(* Logix 5000 project; controller DUNEW2PLC1 vendor 1 type 14 code 221 rev 33.11; software revision 33.00 *)

TASK DUNEWINDER2 (continuous, watchdog 500 ms) : main, state_9_unservo, state_11_eot_trip, state_10_error, state_6_latch, state_3_move_xy, state_5_move_z, state_1_ready, tension_pid, queued_motion, state_12_move_xz, state_13_move_yz, state_14_hmi_stop
TASK SafetyTask (periodic, rate 20 ms, priority 10, watchdog 20 ms) : Safety

MODULES
   Local : vendor 1 type 14 code 221 (5069 0, rev 33.11)
      DUNEW2AMP : 2198-P031 (Ethernet 192.168.140.15, rev 11.3, A_MotionDiagnostics RPI 1 ms, B_MotionSync RPI 2 ms)
      DUNEW2SERVO1 : vendor 1 type 45 code 31 (Ethernet 192.168.140.16, rev 11.3, C_Safety_Output RPI 20 ms, A_MotionDiagnostics RPI 1 ms, D_Safety_Input RPI 10 ms, B_MotionSync RPI 2 ms)
      DUNEW2SERVO2 : vendor 1 type 45 code 31 (Ethernet 192.168.140.17, rev 11.2, A_MotionDiagnostics RPI 1 ms, C_Safety_Output RPI 20 ms, B_MotionSync RPI 2 ms, D_Safety_Input RPI 10 ms)
      DUNEW2NETSW : vendor 1 type 12 code 241 (Ethernet 192.168.140.10, rev 10.1, Output RPI 1000 ms)
      DUNE2CAM1 : vendor 678 type 100 code 274 (Ethernet 192.168.140.19, rev 11.1, Output RPI 60 ms)
       : 5069-IB16 (5069 1, rev 2.14, StandardDataDriven RPI 5 ms)
           Local:1:I.Pt15.Data   // The wire break switch was causing electrical problems, so we use the load-cell as a proxy for wire break
           Local:1:I.Pt09.Data   // Latch middle
           Local:1:I.Pt08.Data   // Latch top
       : 5069-IB16 (5069 6, rev 2.14, StandardDataDriven RPI 5 ms)
       : 5069-IB16 (5069 2, rev 2.14, StandardDataDriven RPI 5 ms)
           Local:2:I.Pt07.Data   // O/T SWITCH OVERTRAVEL SWITCH
           Local:2:I.Pt13.Data   // Cabinet lighted push button
           Local:2:I.Pt06.Data   // TENSION ON/OFF
       : vendor 1 type 115 code 313 (5069 5, rev 2.1, StandardDataDriven RPI 13.1 ms)
           Local:5:O.Ch00.Data   // Tension_Servo_CMD
       : 5069-OB16 (5069 3, rev 2.14, StandardDataDriven RPI 5 ms)
           Local:3:O.Pt01.Data   // Latching signal output
           Local:3:O.Pt11.Data   // Reset PB - Light
           Local:3:O.Pt15.Data   // Beacon - Sounder
           Local:3:O.Pt13.Data   // Beacon - Amber
           Local:3:O.Pt14.Data   // Beacon - Red
           Local:3:O.Pt12.Data   // Beacon - Green
       : 5069-OB16 (5069 7, rev 2.14, StandardDataDriven RPI 5 ms)
       : 5069-IF8 (5069 4, rev 2.11, StandardDataDriven RPI 12.5 ms)
           Local:4:I   // Wire tension (N)
      DUNEW2PLC2 : 1734-AENT (Ethernet 192.168.140.14, rev 6.12)
          : vendor 1 type 35 code 16 (PointIO 2, rev 2.1, Output RPI 20 ms, Input RPI 10 ms)
          : vendor 1 type 35 code 15 (PointIO 1, rev 2.1, Output RPI 20 ms, Input RPI 10 ms)
              DUNEW2PLC2:1:I.Pt03Data   // EStop Pullcord 1
              DUNEW2PLC2:1:I.Pt01Data   // LC OSS2
              DUNEW2PLC2:1:I.Pt00Data   // LC OSS1
              DUNEW2PLC2:1:I.Pt04Data   // EStop Pullcord 2
              DUNEW2PLC2:1:I.Pt02Data   // EStop Rack
              DUNEW2PLC2:1:I.Pt05Data   // Run Key
END_MODULES

TYPE MotionSeg :   // motion segments for move queue, lines or arcs
STRUCT
   Valid : BOOL;   // segment valid flag
   SegType : SINT;   // 1=line, 2=arc
   XY : REAL[2];   // end xy
   Speed : REAL;   // >0
   Accel : REAL;   // >0
   Decel : REAL;   // >0
   JerkAccel : REAL;
   JerkDecel : REAL;
   TermType : SINT;   // 0 to 6
   Seq : DINT;   // Sequence/ack id
   CircleType : DINT;   // 0,1,2,3 per MCCM enum
   ViaCenter : REAL[2];   // [0]=x [1]=y
   Direction : DINT;   // 0..3 per mmcm enum
END_STRUCT
END_TYPE

ADD_ON_INSTRUCTION SCP   (* revision 1.0, vendor CVKI *)
// Scale with Parameters
// Help:
// Rockwell Software RSLogix 500 Description:
// The Input value is scaled to a range determined by creating a linear relationship between input min and max values and scaled min and max values. The scaled result is returned to the address indicated by the output parameter.
VAR_INPUT
   Input : REAL; {required}   // Value to be Scaled
   Input_Min : REAL; {required}   // Minimum Value for the Input
   Input_Max : REAL; {required}   // Maximum Value for the Input
   Scaled_Min : REAL; {required}   // Minimum Scaling Value
   Scaled_Max : REAL; {required}   // Maximum Scaling Value
END_VAR
VAR_OUTPUT
   Output : REAL; {access Read Only, required}   // Scaled Value [Slope*Input + Offset]
END_VAR
VAR
   offset : REAL;   // Offset Value [Scaled Min - (Input Min * Slope)]
   slope : REAL;   // Slope Value [(Scaled Max - Scaled Min)/(Input Max - Input Min)]
END_VAR

ROUTINE Logic   (* ladder *)
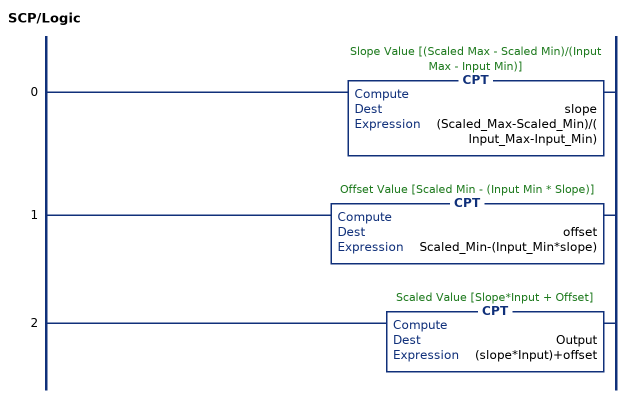
   0: CPT(slope,(Scaled_Max-Scaled_Min)/(Input_Max-Input_Min));
   1: CPT(offset,Scaled_Min-(Input_Min*slope));
   2: CPT(Output,(slope*Input)+offset);
END_ROUTINE
END_ADD_ON_INSTRUCTION

VAR_GLOBAL   (* controller tags *)
   AbortQueue : BOOL;
   accel_xy : REAL;   // Tangential acceleration of the winding head in xy-plane
   ActiveSeq : DINT;
   ACTUATOR_POS : DINT := 2; {access Read Only}
   ALL_EOT_GOOD : BOOL := 1; {access Read Only}
   APA_IS_VERTICAL : BOOL := 1; {access Read Only}
   blink_off : TIMER := (PRE := 500);
   blink_on : TIMER := (PRE := 500, ACC := 98, EN := 1, TT := 1);
   btm_support_collision_ymax : DINT := 440; {access Read Only}
   btm_support_collision_ymin : DINT := 80; {access Read Only}
   CAM_F_EN : BOOL := 1;
   CAM_F_TRIGGER : BOOL := 1;
   check_tension_stable : BOOL := 1;   // Check if the tension is stable at the setpoint before moving the winding head
   CurIssueAckTON : TIMER := (PRE := 100);
   CurIssued : BOOL;
   current_command : REAL := 0.63393843;
   current_command_high : REAL := 1.5; {constant}
   current_command_low : REAL := -0.5; {constant}
   delay_mid_position : TIMER := (PRE := 200, ACC := 200, EN := 1, DN := 1);
   DUNEW1AMP : AXIS_CIP_DRIVE;
   DUNEW2AXIS : MOTION_GROUP;
   EN_POS_TRIGGERS : BOOL;
   ENABLE_ACTUATOR : BOOL;
   Enable_SFX : BOOL;
   Enable_SLS : BOOL;
   ERROR_CODE : DINT; {access Read Only}
   ESTOP : ALIAS FOR DUNEW2PLC2:1:I.Pt02Data;
   FIFO_Data : REAL[6]; {access Read Only}
   FIFO_FLUSH : BOOL;   // Flush the camera FIFOs.
   FRAME_LOC_FT_BTM : BOOL;
   FRAME_LOC_FT_MID : BOOL := 1;
   FRAME_LOC_FT_TOP : BOOL := 1;
   FRAME_LOC_HD_BTM : BOOL;
   FRAME_LOC_HD_MID : BOOL := 1;
   FRAME_LOC_HD_TOP : BOOL := 1;
   gamma : REAL := 2411.3965;
   gui_stop : MOTION_INSTRUCTION := (FLAGS := 33554432);
   HEAD_POS : DINT := 3;
   HomeTrigger : BOOL;
   IncomingSeg : MotionSeg := (Valid := 1, SegType := 1, XY[0] := 2787.4907, Speed := 600.0, Accel := 2000.0, Decel := 2000.0, JerkAccel := 1500.0, JerkDecel := 1500.0, Seq := 1037, CircleType := 1, Direction := 1);
   IncomingSegAck : DINT := 1037;
   IncomingSegReqID : DINT := 4861;
   INIT_DONE : BOOL := 1; {access Read Only}
   J : REAL := 2000.0;
   LastIncomingSegReqID : DINT := 4861;
   LATCH_ACTUATOR_HOMED : BOOL; {access Read Only}
   LATCH_ACTUATOR_MID : BOOL := 1;
   LATCH_ACTUATOR_TOP : BOOL := 1;
   latching_in_progress : BOOL; {access Read Only}
   MACHINE_SW_STAT : BOOL[32] := ([7] := 1, [8] := 1, [10] := 1, [12] := 1, [13] := 1, [14] := 1, [15] := 1, [18] := 1, [19] := 1, [20] := 1, [21] := 1, [22] := 1, [25] := 1, [26] := 1, [27] := 1, [29] := 1, [30] := 1); {access Read Only}
   MASTER_Z_GO : BOOL := 1; {access Read Only}
   max_tolerable_tension : REAL := 9.5;
   MAX_TOLERABLE_Z : REAL := 5.0; {constant}
   MCCD_X_Y_Axis : MOTION_INSTRUCTION := (FLAGS := 301989888, ER := 1, ERR := 5, EXERR := 1);
   MCCD_X_Y_Axis1 : MOTION_INSTRUCTION := (FLAGS := 33554432);
   MCD1_X_axis : MOTION_INSTRUCTION := (FLAGS := -1845493760, EN := 1, ER := 1, ERR := 19);
   MCD_X_axis : MOTION_INSTRUCTION := (FLAGS := 33554432);
   mid_support_collision_ymax : DINT := 1515; {access Read Only}
   mid_support_collision_ymin : DINT := 1050; {access Read Only}
   MINUS_X_EOT : BOOL := 1; {access Read Only}
   MINUS_Y_EOT : BOOL := 1; {access Read Only}
   MORE_STATS : BOOL[32]; {access Read Only}
   MORE_STATS_S : BOOL[32] := ([0] := 1);
   MotionFault : BOOL;
   MOVE_TYPE : INT;   // 0 = No Move 1 = XY JOG 2 = XY Plane Move 3 = Z JOG 4 = Z Axis Move 5 = Toggle Latch Actuator 6 = Home the Latch Actuator 7 = Unlock Latch Actuator Motor 8 = Un-Servo Motors 9 = PLC_Init
   neutral_cv : REAL := 2.5;
   NextIssueAckTON : TIMER := (PRE := 100);
   NextIssued : BOOL;
   NEXTSTATE : DINT := 5; {access Read Only}
   no_apa_collision : BOOL := 1;
   no_latch_collision : BOOL := 1;
   no_supports_collision : BOOL := 1;
   overtension_timer : TIMER := (PRE := 25);
   PendingSeq : DINT;
   pid_cv_high_limit : REAL := 10.0;
   pid_cv_low_limit : REAL;
   PID_LOOP_TIMER : TIMER := (PRE := 3, ACC := 2, EN := 1, TT := 1);
   PLUS_X_EOT : BOOL := 1; {access Read Only}
   PLUS_Y_EOT : BOOL := 1; {access Read Only}
   POSITION : REAL[1,2] := ([0,0] := 7170.4, [0,1] := 309.48557);
   QueueCount : DINT;
   QueueDiag_AbortActive : BOOL;
   QueueDiag_ActiveSeq : DINT;
   QueueDiag_CheckCurSeg : BOOL;
   QueueDiag_CheckNextSeg : BOOL;
   QueueDiag_CmdA_SegType : DINT := 1;
   QueueDiag_CmdB_SegType : DINT := 1;
   QueueDiag_CurSeg_SegType : DINT := 1;
   QueueDiag_CurSeg_Seq : DINT;
   QueueDiag_CurSeg_Speed : DINT := 600;
   QueueDiag_CurSeg_TermType : DINT;
   QueueDiag_CurSeg_Valid : BOOL;
   QueueDiag_CurSeg_X : DINT := 6345;
   QueueDiag_CurSeg_Y : DINT := 2683;
   QueueDiag_FaultCode : DINT;
   QueueDiag_FlipToA : BOOL;
   QueueDiag_FlipToB : BOOL;
   QueueDiag_IssueCurPulse : BOOL;
   QueueDiag_IssueNextPulse : BOOL;
   QueueDiag_LoadCurReq : BOOL;
   QueueDiag_LoadNextReq : BOOL;
   QueueDiag_MoveA_DN : BOOL;
   QueueDiag_MoveA_ER : BOOL;
   QueueDiag_MoveA_ERRID : DINT;
   QueueDiag_MoveA_EXERR : DINT;
   QueueDiag_MoveA_IP : BOOL;
   QueueDiag_MoveA_PC : BOOL;
   QueueDiag_MoveB_DN : BOOL;
   QueueDiag_MoveB_ER : BOOL;
   QueueDiag_MoveB_ERRID : DINT;
   QueueDiag_MoveB_EXERR : DINT;
   QueueDiag_MoveB_IP : BOOL;
   QueueDiag_MoveB_PC : BOOL;
   QueueDiag_NextSeg_SegType : DINT := 1;
   QueueDiag_NextSeg_Seq : DINT;
   QueueDiag_NextSeg_Speed : DINT := 600;
   QueueDiag_NextSeg_TermType : DINT;
   QueueDiag_NextSeg_Valid : BOOL;
   QueueDiag_NextSeg_X : DINT := 5807;
   QueueDiag_NextSeg_Y : DINT := 2683;
   QueueDiag_PendingSeq : DINT;
   QueueDiag_PrepCurMove : BOOL;
   QueueDiag_PrepNextMove : BOOL;
   QueueDiag_QueueCtl_DN : BOOL;
   QueueDiag_QueueCtl_EM : BOOL := 1;
   QueueDiag_QueueCtl_EN : BOOL;
   QueueDiag_QueueCtl_ER : BOOL;
   QueueDiag_QueueCtl_EU : BOOL;
   QueueDiag_QueueCtl_IN : BOOL;
   QueueDiag_QueueCtl_LEN : DINT := 32;
   QueueDiag_QueueCtl_POS : DINT;
   QueueDiag_QueueCtl_UL : BOOL;
   QueueDiag_RotateMoves : BOOL;
   QueueDiag_UseAasCurrent : BOOL := 1;
   QueueDiag_WaitCurAxisOn : BOOL;
   QueueDiag_WaitNextAxisOn : BOOL;
   QueueFault : BOOL;
   QueueFull : BOOL;
   QueueStopRequest : BOOL;
   READ_FIFOS : BOOL;
   ResetPB : BOOL;
   resetPB_S : BOOL;
   ROT_LOC_KEY : AB:1769_DI32:I:0; {access Read Only}
   Run_Alarm : BOOL;
   Safety_Reset_FallingEdge : BOOL;
   Safety_System_Healthy : BOOL := 1;
   Safety_Tripped_S : BOOL;
   SegQueue : MotionSeg[32];
   SLS_Active_Limit : REAL := 50.0;
   SLS_Request1 : BOOL;
   speed_regulator_switch : BOOL := 1;   // This is our "enable safe speed" switch, repurposed to switch the speed regulator
   StartQueuedPath : BOOL;
   STATE : DINT := 5; {access Read Only}   // CURRENT State Machine State
   STATE_FAULT_FLAGS : DINT;
   STATE_REQUEST : DINT := 5;
   STATE_REQUEST_ACK : DINT;
   STATE_REQUEST_ID : DINT;
   STATE_REQUEST_RESULT : DINT := 1;
   support_collision_window_bttm : BOOL := 1;
   support_collision_window_mid : BOOL;
   support_collision_window_top : BOOL;
   T01 : TIMER := (PRE := 5000, ACC := 5000, EN := 1, DN := 1);
   tension : REAL := 6.31352;   // wire tension from load cell (N)
   TENSION_CONTROL_OK : BOOL := 1;
   tension_motor_curr_override : REAL := 6.0;
   tension_motor_cv : REAL := 5.663237;
   tension_off_oneshot : BOOL;
   tension_on_oneshot : BOOL;
   TENSION_ON_SWITCH : BOOL := 1;
   tension_on_switch_delay_on_start : TIMER := (PRE := 500, ACC := 500, EN := 1, DN := 1);
   tension_setpoint : REAL := 6.5;
   tension_stable_timer : TIMER := (PRE := 10);
   tension_tag : ALIAS FOR Local:4:I.Ch01.Data;   // wire tension (N)
   top_support_collision_ymax : DINT := 2650; {access Read Only}
   top_support_collision_ymin : DINT := 2200; {access Read Only}
   v_0 : REAL := 716.5472;
   v_x_max : DINT := 825; {constant, access Read Only}
   v_xy : REAL := 0.3041381;   // velocity of winding head in xy plane
   v_xyz : REAL := 709.44995;   // Velocity of winding head in xyz space
   v_y_max : DINT := 600; {constant, access Read Only}
   winding_head_pid : PID := (CTL := 134251008, DOE := 1, INI := 1, DVPA := 1, SP := 6.5, KI := 0.3, BIAS := 25.0, MAXS := 11.0, SO := 57.91839, MAXO := 100.0, UPD := 0.03, PV := 6.339531, ERR := 0.16046906, OUT := 57.91839, PVH := 10.0, MAXI := 11.0, MAXCV := 10.0, MAXTIE := 10.0, DATA[0] := 32.91839, DATA[1] := 23.340954, DATA[2] := 6.339531, DATA[3] := 0.16046906, DATA[4] := 6.5, DATA[5] := 9.090909, DATA[6] := 1.0, DATA[7] := 0.48, DATA[9] := 0.3, DATA[12] := 0.3, DATA[15] := 0.1, DATA[16] := 10.0);
   wire_broken_tension : REAL := 1.0;
   wire_tensioned : BOOL := 1;
   X_axis : AXIS_CIP_DRIVE; {access Read Only}
   X_Axis_SFX : SAFETY_FEEDBACK_INTERFACE := (FeedbackValid := 1, O1 := 1, PositionScaling := 512.0, FeedbackResolution := 512, Unwind := 512, FeedbackPosition := -428278, ActualPosition := 0.51953125, ActualCycles := -837, FaultType := 1, PositionScalingOut := 512.0, UnwindOut := 512);
   X_Axis_SLS : SAFELY_LIMITED_SPEED := (RestartType := 1, ColdStartType := 1, O1 := 1, CheckDelay := 3000, ActiveLimit := 10.0, FaultType := 1);
   X_DELTA : REAL;
   X_PARKED : BOOL := 1; {access Read Only}
   X_POSITION : ALIAS FOR POSITION[0,0];
   X_XFER_OK : BOOL := 1; {access Read Only}   // If at the head, check head support arms. Same for foot
   X_Y : COORDINATE_SYSTEM;
   XY_ACCELERATION : REAL := 2000.0;   // Maximum positive acceleration for position move.
   XY_DECELERATION : REAL := 2000.0;   // Maximum negative acceleration for position move.
   xy_regulated_acceleration : REAL := 2000.0;
   xy_regulated_deceleration : REAL := 2000.0;
   XY_SPEED : REAL := 300.0;   // Maximum velocity for position move.
   XY_SPEED_REQ : REAL := 300.0;   // XY Requested speed copy of XY_Speed to be used for MCLM and MCCD in MoveXY
   xyz : COORDINATE_SYSTEM;
   xz : COORDINATE_SYSTEM;
   xz_position_target : REAL[2] := ([0] := 6000.0);
   xz_speed : DINT := 300;
   Y_axis : AXIS_CIP_DRIVE; {access Read Only}
   Y_DELTA : REAL := 5.75;
   Y_MOUNT_XFER_OK : BOOL; {access Read Only}
   Y_POSITION : ALIAS FOR POSITION[0,1];
   Y_XFER_OK : BOOL; {access Read Only}
   yz : COORDINATE_SYSTEM;
   yz_position_target : REAL[2] := ([0] := 119.9572, [1] := -0.0016);
   yz_speed : DINT := 100;
   Z_ACCELERATION : REAL := 2000.0;
   Z_axis : AXIS_CIP_DRIVE; {access Read Only}
   Z_DECELLERATION : REAL := 2000.0;
   Z_EOT : BOOL := 1; {access Read Only}
   z_eot_bypass : BOOL := 1;
   Z_EXTENDED : BOOL; {access Read Only}
   Z_FIXED_LATCHED : BOOL := 1; {access Read Only}
   Z_FIXED_PRESENT : BOOL := 1; {access Read Only}
   Z_POSITION : REAL;
   Z_RETRACTED : BOOL; {access Read Only}
   Z_SPEED : REAL := 300.0;
   Z_STAGE_LATCHED : BOOL; {access Read Only}
   Z_STAGE_PRESENT : BOOL; {access Read Only}   // Winding head is on the Z-arm
END_VAR

PROGRAM Camera   (* main routine CameraControl *)
// Controls to capture data from the Cognex camera.
VAR
   Cam_F_InspectionRes_0 : REAL[32]; {access Read Only}
   Cam_F_InspectionRes_1 : REAL[10]; {access Read Only}
   Cam_F_InspectionRes_2 : REAL[10]; {access Read Only}
   Cam_F_InspectionRes_3 : REAL[10]; {access Read Only}
   FIFO_CTRL : CONTROL[6] := ([0].LEN := 10, [0].EM := 1, [1].LEN := 10, [1].EM := 1, [2].LEN := 10, [2].EM := 1, [3].LEN := 10, [3].EM := 1, [4].LEN := 10, [4].EM := 1, [5].LEN := 10, [5].EM := 1); {access Read Only}
   foundIt : BOOL; {access Read Only}
   LightRing : TIMER := (PRE := 100); {access Read Only}
   Manual_Trig : BOOL; {access Read Only}
   osob : BOOL[32]; {access Read Only}
   ossb : BOOL[32] := ([3] := 1); {access Read Only}
   Pos_trigger : BOOL := 1; {access Read Only}
   RegistrationData : MOTION_INSTRUCTION[8] := ([0].FLAGS := -1845493760, [0].EN := 1, [0].ER := 1, [0].ERR := 3, [1].FLAGS := -1845493760, [1].EN := 1, [1].ER := 1, [1].ERR := 3); {access Read Only}
   test_tag : BOOL;   // Demo tag added to show how Studio creates new tags on routine import
   triggerOneShotOB : BOOL; {access Read Only}
   triggerOneShotSB : BOOL := 1; {access Read Only}
   TriggerResetTimer1 : TIMER := (PRE := 100, ACC := 5, EN := 1, TT := 1); {access Read Only}
   TriggerResetTimer2 : TIMER := (PRE := 100); {access Read Only}
   X_axis_Cam_F_Pos : REAL[10]; {access Read Only}
   X_axis_Cam_F_Position : REAL := -5.1799655; {access Read Only}
   x_pos : REAL := 564.005; {access Read Only}
   x_pos_next : REAL := 564.005;
   Y_axis_Cam_F_Pos : REAL[10]; {access Read Only}
   Y_axis_Cam_F_Position : REAL := 12.123628; {access Read Only}
   y_pos : REAL := 2465.8398;
   y_pos_next : REAL := 2465.8398;
   Z_RETRACTED_1A : BOOL := 1; {access Read Only}
   Z_RETRACTED_1B : BOOL := 1; {access Read Only}
   Z_RETRACTED_2A : BOOL := 1; {access Read Only}
   Z_RETRACTED_2B : BOOL := 1; {access Read Only}
END_VAR

ROUTINE CameraControl   (* ladder *)
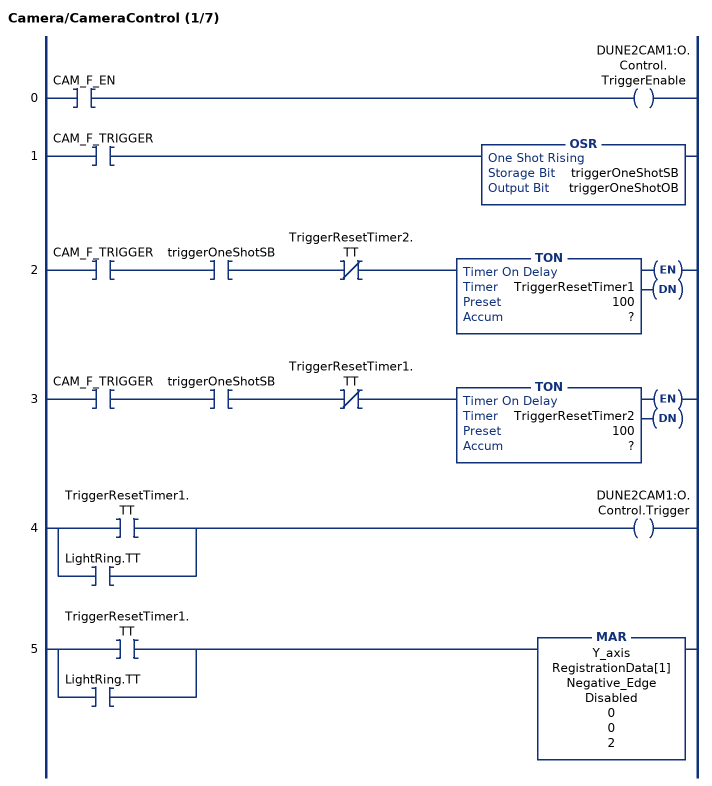
   0: XIC(CAM_F_EN)OTE(DUNE2CAM1:O.Control.TriggerEnable);
   1: XIC(CAM_F_TRIGGER)OSR(triggerOneShotSB,triggerOneShotOB);
   2: XIC(CAM_F_TRIGGER)XIC(triggerOneShotSB)XIO(TriggerResetTimer2.TT)TON(TriggerResetTimer1,?,?);
   3: XIC(CAM_F_TRIGGER)XIC(triggerOneShotSB)XIO(TriggerResetTimer1.TT)TON(TriggerResetTimer2,?,?);
   4: [XIC(TriggerResetTimer1.TT) ,XIC(LightRing.TT) ]OTE(DUNE2CAM1:O.Control.Trigger);
   5: [XIC(TriggerResetTimer1.TT) ,XIC(LightRing.TT) ]MAR(Y_axis,RegistrationData[1],Negative_Edge,Disabled,0,0,2);
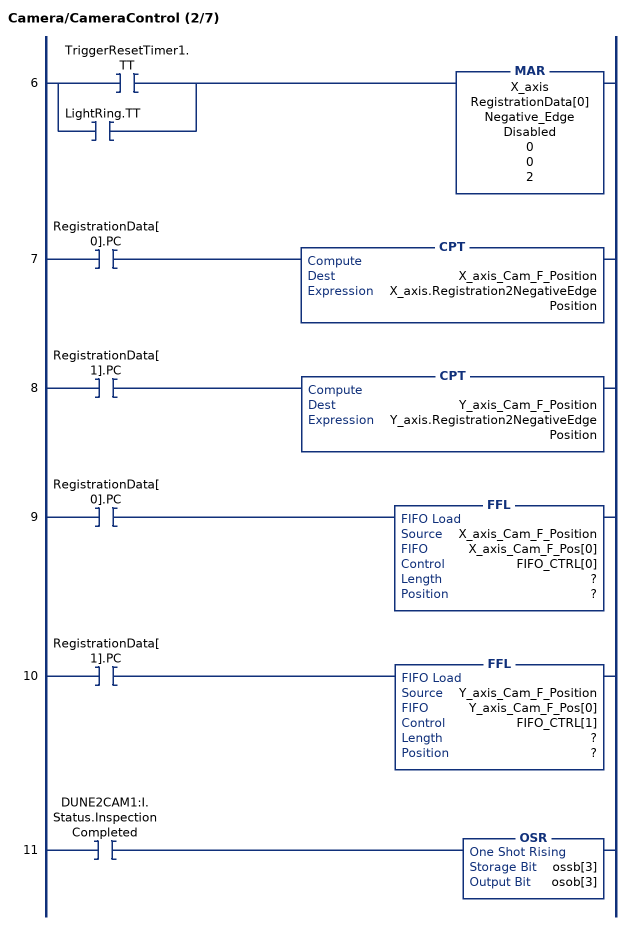
   6: [XIC(TriggerResetTimer1.TT) ,XIC(LightRing.TT) ]MAR(X_axis,RegistrationData[0],Negative_Edge,Disabled,0,0,2);
   7: XIC(RegistrationData[0].PC)CPT(X_axis_Cam_F_Position,X_axis.Registration2NegativeEdgePosition);
   8: XIC(RegistrationData[1].PC)CPT(Y_axis_Cam_F_Position,Y_axis.Registration2NegativeEdgePosition);
   9: XIC(RegistrationData[0].PC)FFL(X_axis_Cam_F_Position,X_axis_Cam_F_Pos[0],FIFO_CTRL[0],?,?);
   10: XIC(RegistrationData[1].PC)FFL(Y_axis_Cam_F_Position,Y_axis_Cam_F_Pos[0],FIFO_CTRL[1],?,?);
   11: XIC(DUNE2CAM1:I.Status.InspectionCompleted)OSR(ossb[3],osob[3]);
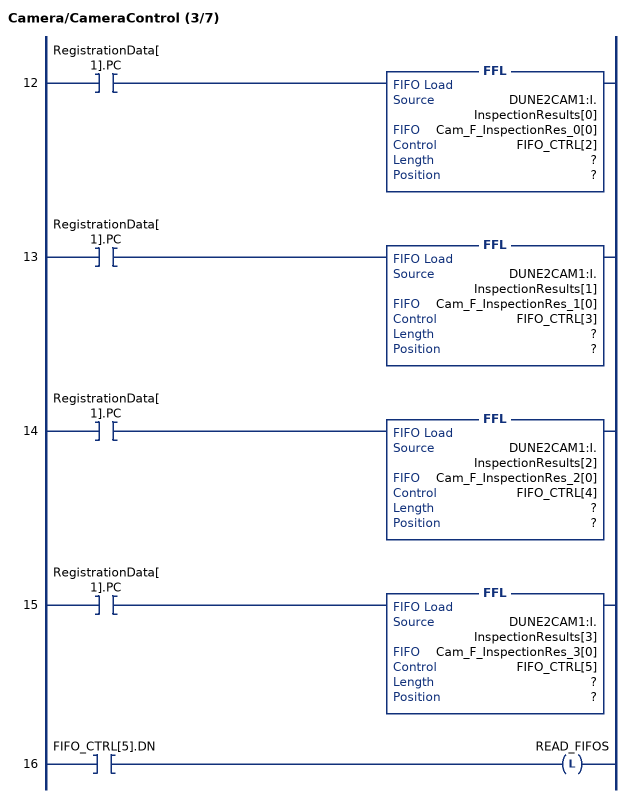
   12: XIC(RegistrationData[1].PC)FFL(DUNE2CAM1:I.InspectionResults[0],Cam_F_InspectionRes_0[0],FIFO_CTRL[2],?,?);
   13: XIC(RegistrationData[1].PC)FFL(DUNE2CAM1:I.InspectionResults[1],Cam_F_InspectionRes_1[0],FIFO_CTRL[3],?,?);
   14: XIC(RegistrationData[1].PC)FFL(DUNE2CAM1:I.InspectionResults[2],Cam_F_InspectionRes_2[0],FIFO_CTRL[4],?,?);
   15: XIC(RegistrationData[1].PC)FFL(DUNE2CAM1:I.InspectionResults[3],Cam_F_InspectionRes_3[0],FIFO_CTRL[5],?,?);
   16: XIC(FIFO_CTRL[5].DN)OTL(READ_FIFOS);
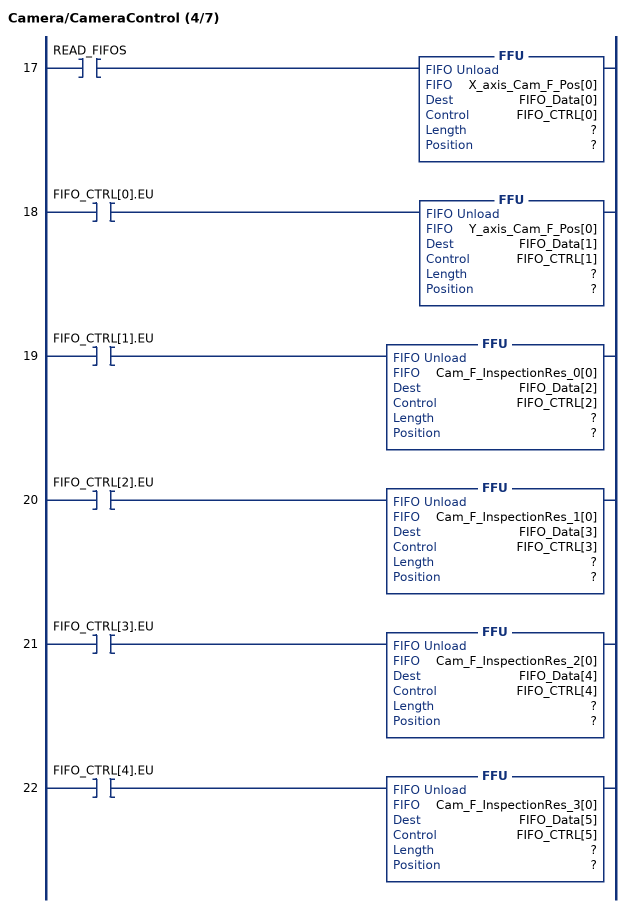
   17: XIC(READ_FIFOS)FFU(X_axis_Cam_F_Pos[0],FIFO_Data[0],FIFO_CTRL[0],?,?);
   18: XIC(FIFO_CTRL[0].EU)FFU(Y_axis_Cam_F_Pos[0],FIFO_Data[1],FIFO_CTRL[1],?,?);
   19: XIC(FIFO_CTRL[1].EU)FFU(Cam_F_InspectionRes_0[0],FIFO_Data[2],FIFO_CTRL[2],?,?);
   20: XIC(FIFO_CTRL[2].EU)FFU(Cam_F_InspectionRes_1[0],FIFO_Data[3],FIFO_CTRL[3],?,?);
   21: XIC(FIFO_CTRL[3].EU)FFU(Cam_F_InspectionRes_2[0],FIFO_Data[4],FIFO_CTRL[4],?,?);
   22: XIC(FIFO_CTRL[4].EU)FFU(Cam_F_InspectionRes_3[0],FIFO_Data[5],FIFO_CTRL[5],?,?);
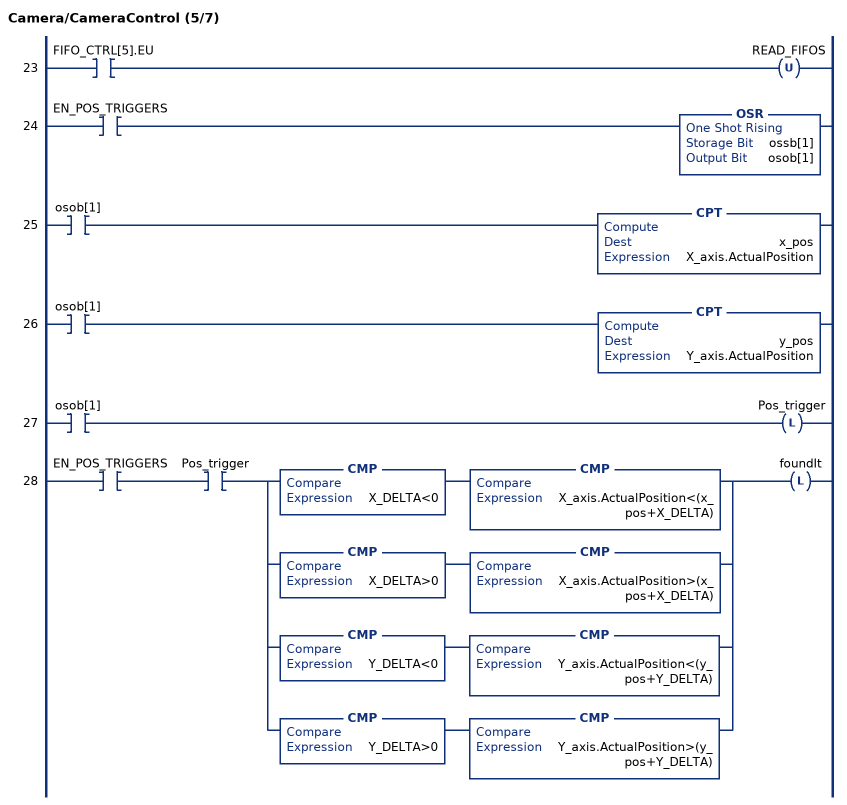
   23: XIC(FIFO_CTRL[5].EU)OTU(READ_FIFOS);
   24: XIC(EN_POS_TRIGGERS)OSR(ossb[1],osob[1]);
   25: XIC(osob[1])CPT(x_pos,X_axis.ActualPosition);
   26: XIC(osob[1])CPT(y_pos,Y_axis.ActualPosition);
   27: XIC(osob[1])OTL(Pos_trigger);
   28: XIC(EN_POS_TRIGGERS)XIC(Pos_trigger)[[CMP(X_DELTA<0) CMP(X_axis.ActualPosition<(x_pos+X_DELTA)) ,CMP(X_DELTA>0) CMP(X_axis.ActualPosition>(x_pos+X_DELTA)) ] ,[CMP(Y_DELTA<0) CMP(Y_axis.ActualPosition<(y_pos+Y_DELTA)) ,CMP(Y_DELTA>0) CMP(Y_axis.ActualPosition>(y_pos+Y_DELTA)) ] ]OTL(foundIt);
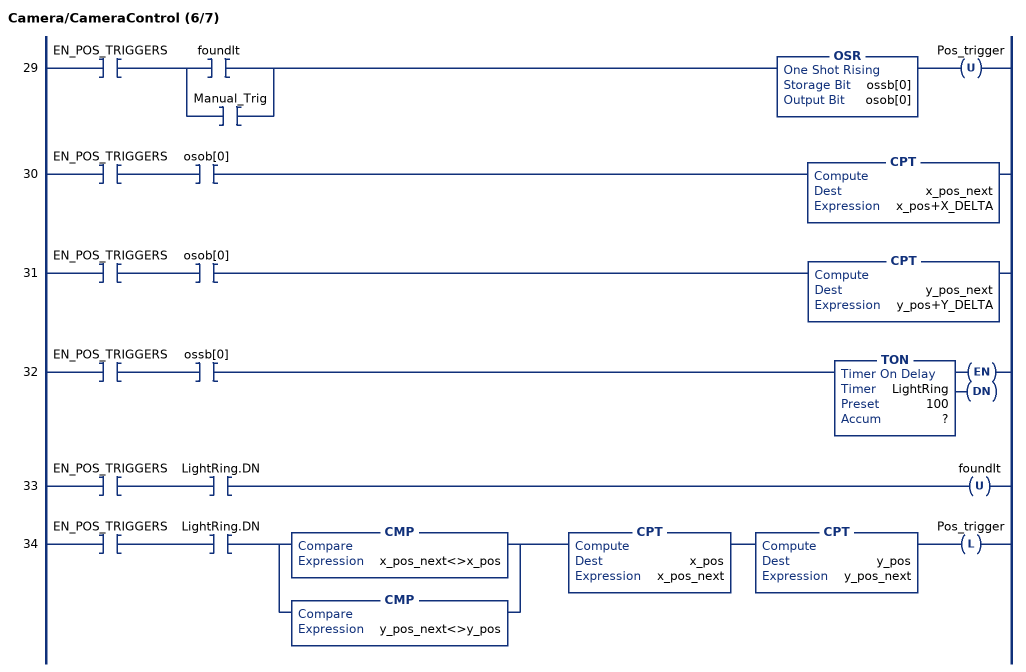
   29: XIC(EN_POS_TRIGGERS)[XIC(foundIt) ,XIC(Manual_Trig) ]OSR(ossb[0],osob[0])OTU(Pos_trigger);
   30: XIC(EN_POS_TRIGGERS)XIC(osob[0])CPT(x_pos_next,x_pos+X_DELTA);
   31: XIC(EN_POS_TRIGGERS)XIC(osob[0])CPT(y_pos_next,y_pos+Y_DELTA);
   32: XIC(EN_POS_TRIGGERS)XIC(ossb[0])TON(LightRing,?,?);
   33: XIC(EN_POS_TRIGGERS)XIC(LightRing.DN)OTU(foundIt);
   34: XIC(EN_POS_TRIGGERS)XIC(LightRing.DN)[CMP(x_pos_next<>x_pos) ,CMP(y_pos_next<>y_pos) ]CPT(x_pos,x_pos_next)CPT(y_pos,y_pos_next)OTL(Pos_trigger);
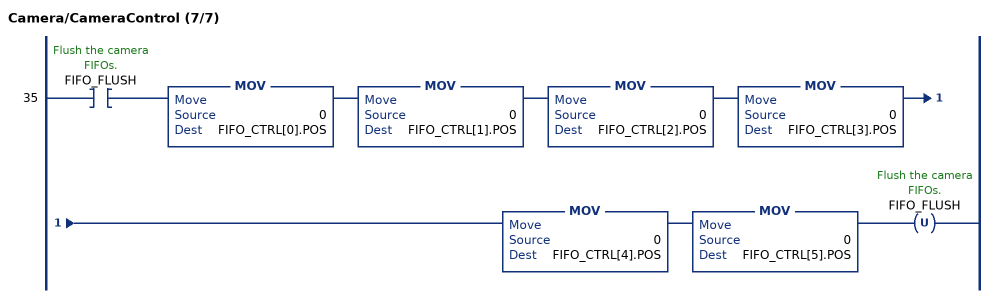
   35: XIC(FIFO_FLUSH)MOV(0,FIFO_CTRL[0].POS)MOV(0,FIFO_CTRL[1].POS)MOV(0,FIFO_CTRL[2].POS)MOV(0,FIFO_CTRL[3].POS)MOV(0,FIFO_CTRL[4].POS)MOV(0,FIFO_CTRL[5].POS)OTU(FIFO_FLUSH);
END_ROUTINE

ROUTINE main   (* ladder *)
END_ROUTINE
END_PROGRAM

PROGRAM main   (* main routine main *)
VAR
   pending_rung_test : BOOL;
   STATE1_IND : BOOL := 1; {access Read Only}
   test_tag : BOOL := 1;   // Demo tag added to show how Studio creates new tags on routine import
   Z_RETRACTED_1A : BOOL; {access Read Only}
   Z_RETRACTED_1B : BOOL; {access Read Only}
   Z_RETRACTED_2A : BOOL; {access Read Only}
   Z_RETRACTED_2B : BOOL; {access Read Only}
END_VAR

ROUTINE main   (* ladder *)
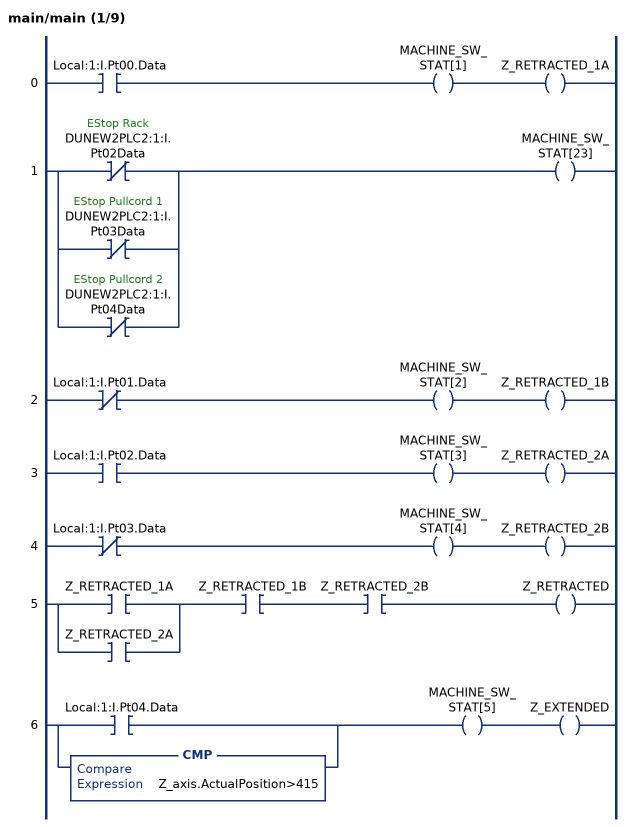
   0: XIC(Local:1:I.Pt00.Data)OTE(MACHINE_SW_STAT[1])OTE(Z_RETRACTED_1A);
   1: [XIO(DUNEW2PLC2:1:I.Pt02Data) ,XIO(DUNEW2PLC2:1:I.Pt03Data) ,XIO(DUNEW2PLC2:1:I.Pt04Data) ]OTE(MACHINE_SW_STAT[23]);
   2: XIO(Local:1:I.Pt01.Data)OTE(MACHINE_SW_STAT[2])OTE(Z_RETRACTED_1B);
   3: XIC(Local:1:I.Pt02.Data)OTE(MACHINE_SW_STAT[3])OTE(Z_RETRACTED_2A);
   4: XIO(Local:1:I.Pt03.Data)OTE(MACHINE_SW_STAT[4])OTE(Z_RETRACTED_2B);
   5: [XIC(Z_RETRACTED_1A) ,XIC(Z_RETRACTED_2A) ]XIC(Z_RETRACTED_1B)XIC(Z_RETRACTED_2B)OTE(Z_RETRACTED);
   6: [XIC(Local:1:I.Pt04.Data) ,CMP(Z_axis.ActualPosition>415) ]OTE(MACHINE_SW_STAT[5])OTE(Z_EXTENDED);
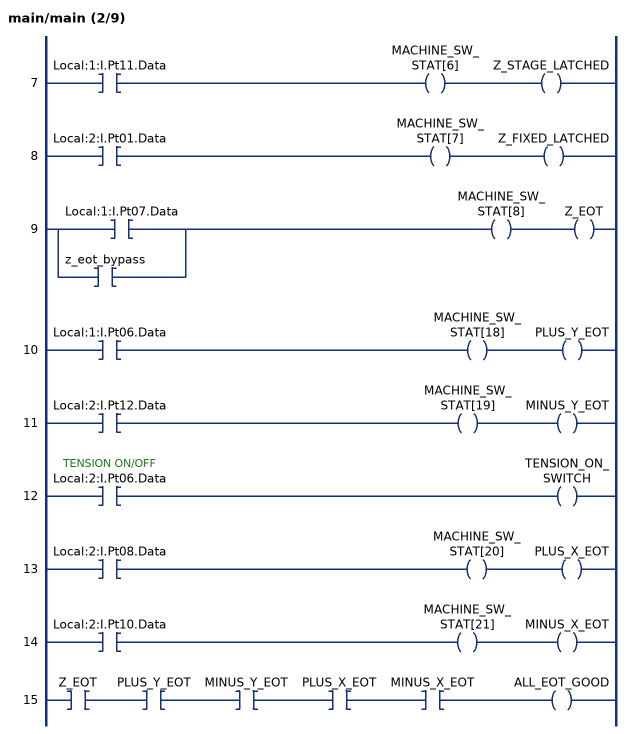
   7: XIC(Local:1:I.Pt11.Data)OTE(MACHINE_SW_STAT[6])OTE(Z_STAGE_LATCHED);
   8: XIC(Local:2:I.Pt01.Data)OTE(MACHINE_SW_STAT[7])OTE(Z_FIXED_LATCHED);
   9: [XIC(Local:1:I.Pt07.Data) ,XIC(z_eot_bypass) ]OTE(MACHINE_SW_STAT[8])OTE(Z_EOT);
   10: XIC(Local:1:I.Pt06.Data)OTE(MACHINE_SW_STAT[18])OTE(PLUS_Y_EOT);
   11: XIC(Local:2:I.Pt12.Data)OTE(MACHINE_SW_STAT[19])OTE(MINUS_Y_EOT);
   12: XIC(Local:2:I.Pt06.Data)OTE(TENSION_ON_SWITCH);
   13: XIC(Local:2:I.Pt08.Data)OTE(MACHINE_SW_STAT[20])OTE(PLUS_X_EOT);
   14: XIC(Local:2:I.Pt10.Data)OTE(MACHINE_SW_STAT[21])OTE(MINUS_X_EOT);
   15: XIC(Z_EOT)XIC(PLUS_Y_EOT)XIC(MINUS_Y_EOT)XIC(PLUS_X_EOT)XIC(MINUS_X_EOT)OTE(ALL_EOT_GOOD);
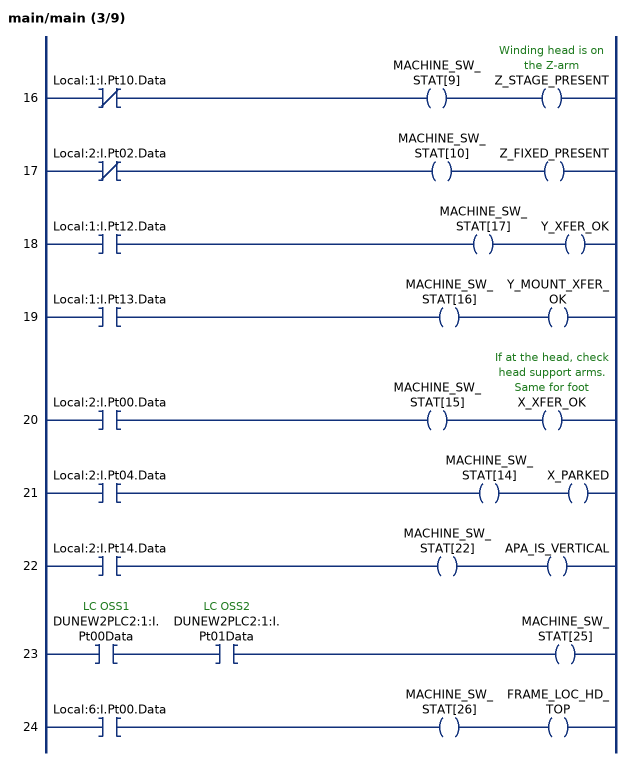
   16: XIO(Local:1:I.Pt10.Data)OTE(MACHINE_SW_STAT[9])OTE(Z_STAGE_PRESENT);
   17: XIO(Local:2:I.Pt02.Data)OTE(MACHINE_SW_STAT[10])OTE(Z_FIXED_PRESENT);
   18: XIC(Local:1:I.Pt12.Data)OTE(MACHINE_SW_STAT[17])OTE(Y_XFER_OK);
   19: XIC(Local:1:I.Pt13.Data)OTE(MACHINE_SW_STAT[16])OTE(Y_MOUNT_XFER_OK);
   20: XIC(Local:2:I.Pt00.Data)OTE(MACHINE_SW_STAT[15])OTE(X_XFER_OK);
   21: XIC(Local:2:I.Pt04.Data)OTE(MACHINE_SW_STAT[14])OTE(X_PARKED);
   22: XIC(Local:2:I.Pt14.Data)OTE(MACHINE_SW_STAT[22])OTE(APA_IS_VERTICAL);
   23: XIC(DUNEW2PLC2:1:I.Pt00Data)XIC(DUNEW2PLC2:1:I.Pt01Data)OTE(MACHINE_SW_STAT[25]);
   24: XIC(Local:6:I.Pt00.Data)OTE(MACHINE_SW_STAT[26])OTE(FRAME_LOC_HD_TOP);
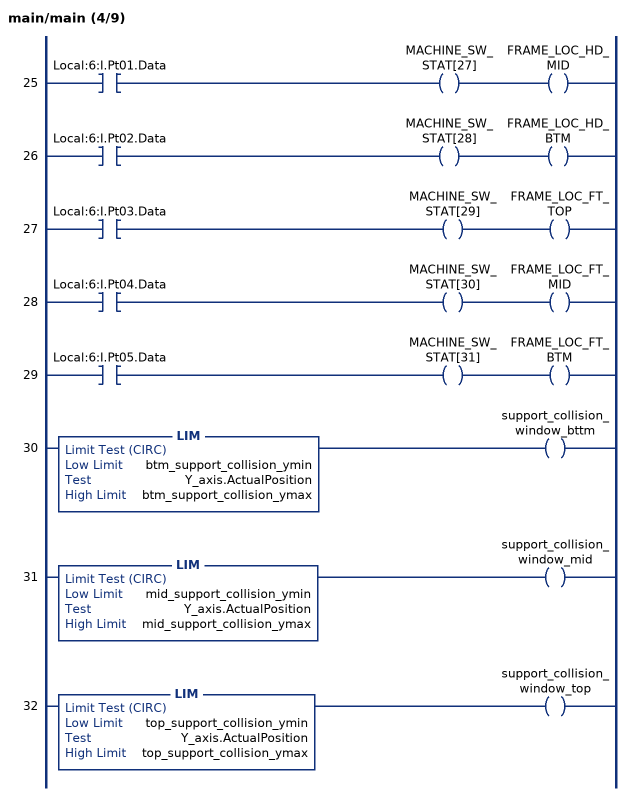
   25: XIC(Local:6:I.Pt01.Data)OTE(MACHINE_SW_STAT[27])OTE(FRAME_LOC_HD_MID);
   26: XIC(Local:6:I.Pt02.Data)OTE(MACHINE_SW_STAT[28])OTE(FRAME_LOC_HD_BTM);
   27: XIC(Local:6:I.Pt03.Data)OTE(MACHINE_SW_STAT[29])OTE(FRAME_LOC_FT_TOP);
   28: XIC(Local:6:I.Pt04.Data)OTE(MACHINE_SW_STAT[30])OTE(FRAME_LOC_FT_MID);
   29: XIC(Local:6:I.Pt05.Data)OTE(MACHINE_SW_STAT[31])OTE(FRAME_LOC_FT_BTM);
   30: LIM(btm_support_collision_ymin,Y_axis.ActualPosition,btm_support_collision_ymax)OTE(support_collision_window_bttm);
   31: LIM(mid_support_collision_ymin,Y_axis.ActualPosition,mid_support_collision_ymax)OTE(support_collision_window_mid);
   32: LIM(top_support_collision_ymin,Y_axis.ActualPosition,top_support_collision_ymax)OTE(support_collision_window_top);
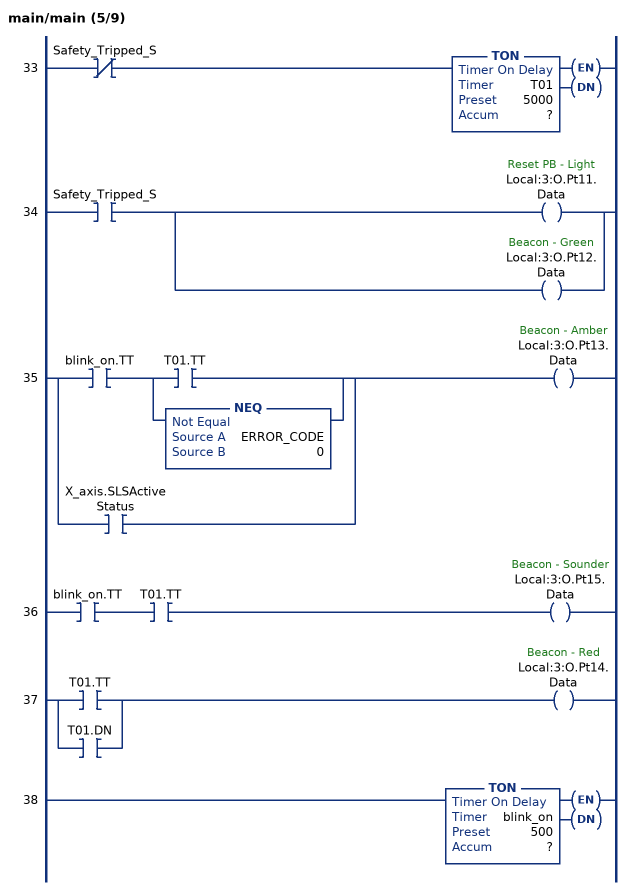
   33: XIO(Safety_Tripped_S)TON(T01,?,?);
   34: XIC(Safety_Tripped_S)[OTE(Local:3:O.Pt11.Data) ,OTE(Local:3:O.Pt12.Data) ];
   35: [XIC(blink_on.TT) [XIC(T01.TT) ,NEQ(ERROR_CODE,0) ] ,XIC(X_axis.SLSActiveStatus) ]OTE(Local:3:O.Pt13.Data);
   36: XIC(blink_on.TT)XIC(T01.TT)OTE(Local:3:O.Pt15.Data);
   37: [XIC(T01.TT) ,XIC(T01.DN) ]OTE(Local:3:O.Pt14.Data);
   38: TON(blink_on,?,?);
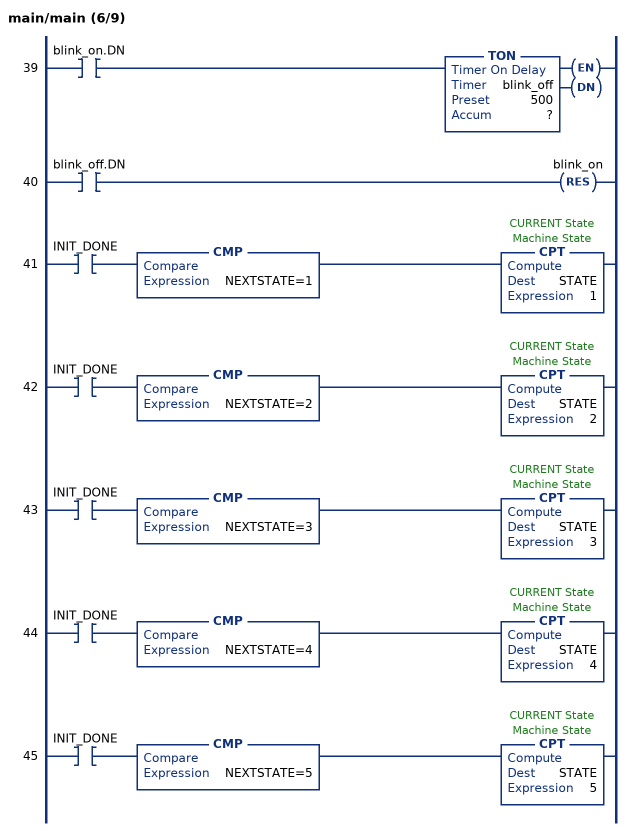
   39: XIC(blink_on.DN)TON(blink_off,?,?);
   40: XIC(blink_off.DN)RES(blink_on);
   41: XIC(INIT_DONE)CMP(NEXTSTATE=1)CPT(STATE,1);
   42: XIC(INIT_DONE)CMP(NEXTSTATE=2)CPT(STATE,2);
   43: XIC(INIT_DONE)CMP(NEXTSTATE=3)CPT(STATE,3);
   44: XIC(INIT_DONE)CMP(NEXTSTATE=4)CPT(STATE,4);
   45: XIC(INIT_DONE)CMP(NEXTSTATE=5)CPT(STATE,5);
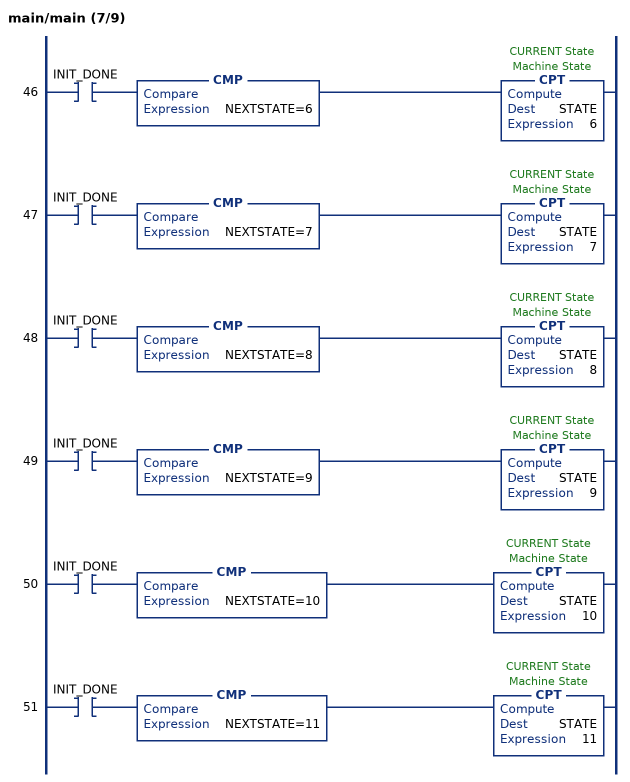
   46: XIC(INIT_DONE)CMP(NEXTSTATE=6)CPT(STATE,6);
   47: XIC(INIT_DONE)CMP(NEXTSTATE=7)CPT(STATE,7);
   48: XIC(INIT_DONE)CMP(NEXTSTATE=8)CPT(STATE,8);
   49: XIC(INIT_DONE)CMP(NEXTSTATE=9)CPT(STATE,9);
   50: XIC(INIT_DONE)CMP(NEXTSTATE=10)CPT(STATE,10);
   51: XIC(INIT_DONE)CMP(NEXTSTATE=11)CPT(STATE,11);
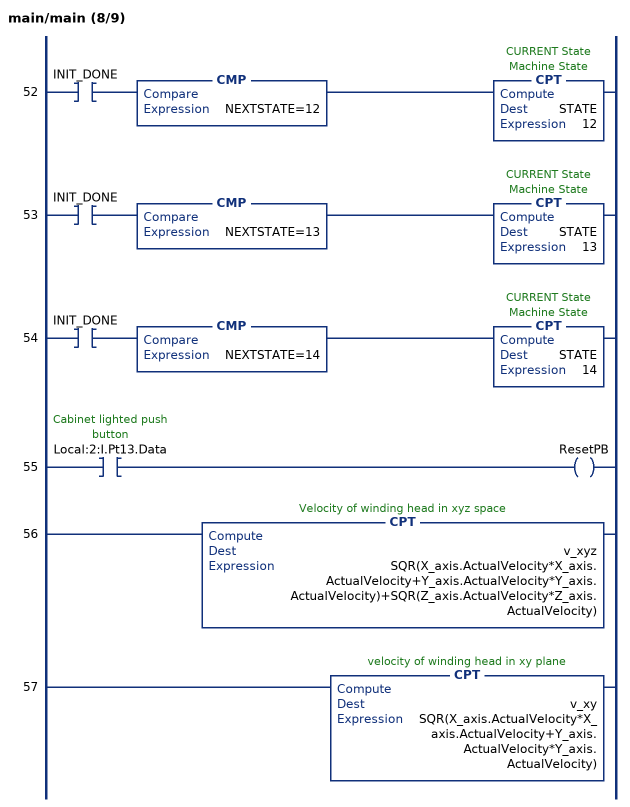
   52: XIC(INIT_DONE)CMP(NEXTSTATE=12)CPT(STATE,12);
   53: XIC(INIT_DONE)CMP(NEXTSTATE=13)CPT(STATE,13);
   54: XIC(INIT_DONE)CMP(NEXTSTATE=14)CPT(STATE,14);
   55: XIC(Local:2:I.Pt13.Data)OTE(ResetPB);
   56: CPT(v_xyz,SQR(X_axis.ActualVelocity*X_axis.ActualVelocity+Y_axis.ActualVelocity*Y_axis.ActualVelocity)+SQR(Z_axis.ActualVelocity*Z_axis.ActualVelocity));
   57: CPT(v_xy,SQR(X_axis.ActualVelocity*X_axis.ActualVelocity+Y_axis.ActualVelocity*Y_axis.ActualVelocity));
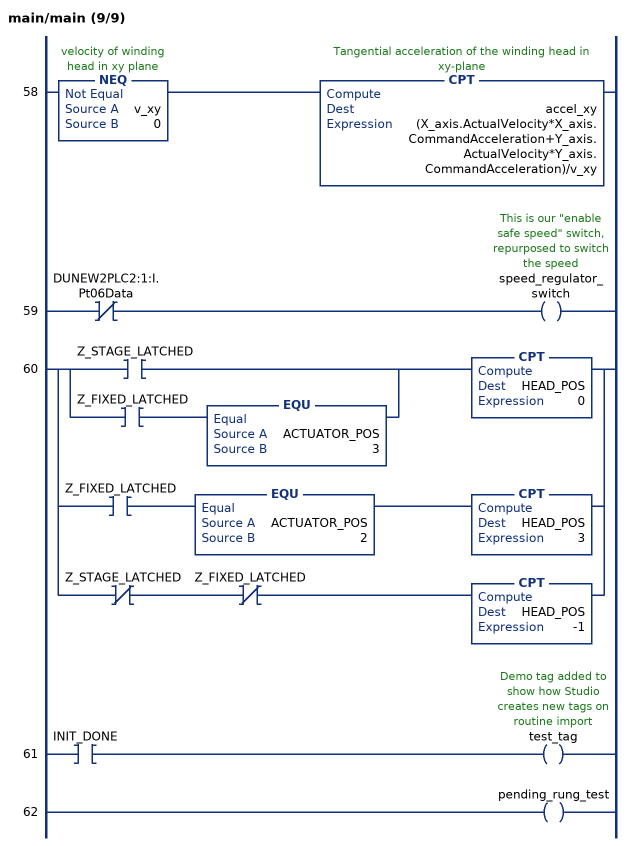
   58: NEQ(v_xy,0)CPT(accel_xy,(X_axis.ActualVelocity*X_axis.CommandAcceleration+Y_axis.ActualVelocity*Y_axis.CommandAcceleration)/v_xy);
   59: XIO(DUNEW2PLC2:1:I.Pt06Data)OTE(speed_regulator_switch);
   60: [[XIC(Z_STAGE_LATCHED) ,XIC(Z_FIXED_LATCHED) EQU(ACTUATOR_POS,3) ] CPT(HEAD_POS,0) ,XIC(Z_FIXED_LATCHED) EQU(ACTUATOR_POS,2) CPT(HEAD_POS,3) ,XIO(Z_STAGE_LATCHED) XIO(Z_FIXED_LATCHED) CPT(HEAD_POS,-1) ];
   61: XIC(INIT_DONE)OTE(test_tag);
   62 (stored rung type 13): OTE(pending_rung_test);
END_ROUTINE
END_PROGRAM

PROGRAM queued_motion   (* main routine main *)
VAR
   AbortActive : BOOL;
   BOOLS : BOOL[1024] := ([7] := 1, [8] := 1, [901] := 1, [902] := 1, [903] := 1);
   CheckCurSeg : BOOL;
   CheckNextSeg : BOOL;
   CmdA_Accel : REAL := 2000.0;
   CmdA_CircleType : DINT := 1;
   CmdA_Decel : REAL := 2000.0;
   CmdA_Direction : DINT := 1;
   CmdA_JerkAccel : REAL := 1500.0;
   CmdA_JerkDecel : REAL := 1500.0;
   CmdA_SegType : DINT := 1;
   CmdA_Speed : REAL := 600.0;
   CmdA_TermType : SINT;
   CmdA_ViaCenter : REAL[2];
   CmdA_XY : REAL[2] := ([0] := 5807.324, [1] := 2683.0);
   CmdB_Accel : REAL := 2000.0;
   CmdB_CircleType : DINT := 1;
   CmdB_Decel : REAL := 2000.0;
   CmdB_Direction : DINT := 1;
   CmdB_JerkAccel : REAL := 1500.0;
   CmdB_JerkDecel : REAL := 1500.0;
   CmdB_SegType : DINT := 1;
   CmdB_Speed : REAL := 600.0;
   CmdB_TermType : SINT;
   CmdB_ViaCenter : REAL[2];
   CmdB_XY : REAL[2] := ([0] := 6344.578, [1] := 2683.0);
   CmdTolerance : DINT := 100;
   CurSeg : MotionSeg := (SegType := 1, XY[0] := 6344.578, XY[1] := 2683.0, Speed := 600.0, Accel := 2000.0, Decel := 2000.0, JerkAccel := 1500.0, JerkDecel := 1500.0, CircleType := 1, Direction := 1);
   DINTS : DINT[1024];
   DoneONS_A : BOOL;
   DoneONS_B : BOOL;
   EnqueueReq : BOOL;
   FaultCode : DINT;
   FlipToA : BOOL;
   FlipToB : BOOL;
   idx_0 : DINT;
   idx_1 : DINT;
   idx_2 : DINT;
   idx_3 : DINT := 1;
   IssueCurPulse : BOOL;
   IssueNextPulse : BOOL;
   LoadCurReq : BOOL;
   LoadNextReq : BOOL;
   MoveA : MOTION_INSTRUCTION := (FLAGS := 33554432);
   MoveB : MOTION_INSTRUCTION := (FLAGS := 33554432);
   NextSeg : MotionSeg := (SegType := 1, XY[0] := 5807.324, XY[1] := 2683.0, Speed := 600.0, Accel := 2000.0, Decel := 2000.0, JerkAccel := 1500.0, JerkDecel := 1500.0, CircleType := 1, Direction := 1);
   PrepCurMove : BOOL;
   PrepNextMove : BOOL;
   QueueCtl : CONTROL := (LEN := 32, EM := 1);
   QueueEmpty : BOOL := 1;
   QueueStopReqONS : BOOL;
   REALS : REAL[1024] := ([14] := 0.17588998, [15] := 0.13223965, [16] := -0.04365033, [17] := 6.2831855, [18] := -0.04365033, [19] := 0.04365033, [20] := 4293.247, [21] := 1201.037, [22] := 0.78177166, [23] := 0.62356484, [24] := -1505.7563, [25] := -1201.037, [26] := 1926.082, [31] := 22.764017, [32] := 27.084085, [33] := 0.17588998, [34] := 0.13223965, [35] := -0.04365033, [38] := 825.0, [39] := 600.0, [40] := 4293.247, [41] := 1201.037, [42] := 2787.4907, [44] := 962.2095, [45] := 0.78177166, [46] := 0.62356484, [47] := 1055.2954, [48] := 962.2095, [49] := 600.0, [910] := -0.04365033, [911] := 0.04365033, [912] := 78.1998, [913] := 440.0006, [914] := 86.11841, [915] := 647.42926);
   RotateMoves : BOOL;
   RotateONS_AtoB : BOOL;
   RotateONS_BtoA : BOOL;
   SegValid : BOOL;
   SegValidArc : BOOL;
   SegValidLine : BOOL;
   StartCurONS : BOOL;
   StartNextA_ONS : BOOL;
   StartNextB_ONS : BOOL;
   UseAasCurrent : BOOL := 1;
   WaitCurAxisOn : BOOL;
   WaitNextAxisOn : BOOL;
   x_axis_mso : MOTION_INSTRUCTION := (FLAGS := 33554432);
   y_axis_mso : MOTION_INSTRUCTION := (FLAGS := 33554432);
END_VAR

ROUTINE ArcSweepRad   (* ladder *)
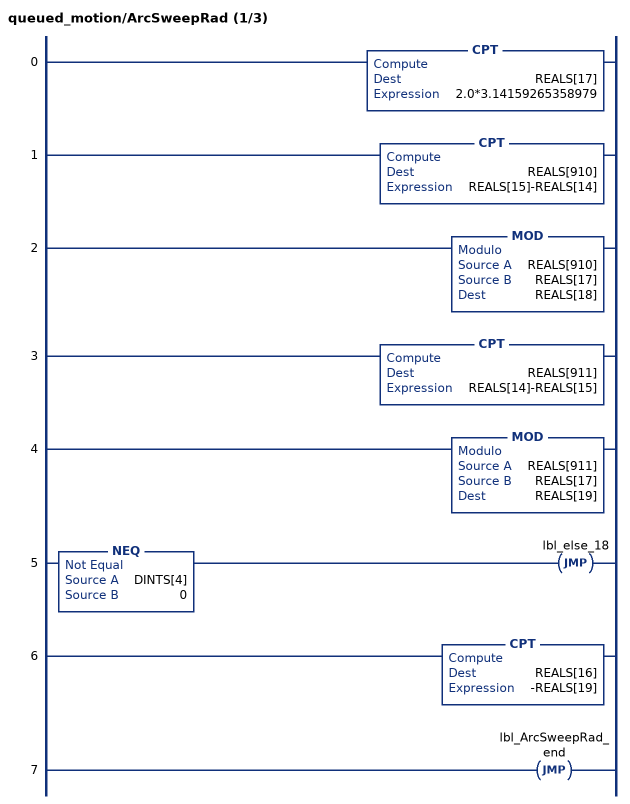
   0: CPT(REALS[17],2.0*3.14159265358979);
   1: CPT(REALS[910],REALS[15]-REALS[14]);
   2: MOD(REALS[910],REALS[17],REALS[18]);
   3: CPT(REALS[911],REALS[14]-REALS[15]);
   4: MOD(REALS[911],REALS[17],REALS[19]);
   5: NEQ(DINTS[4],0)JMP(lbl_else_18);
   6: CPT(REALS[16],-REALS[19]);
   7: JMP(lbl_ArcSweepRad_end);
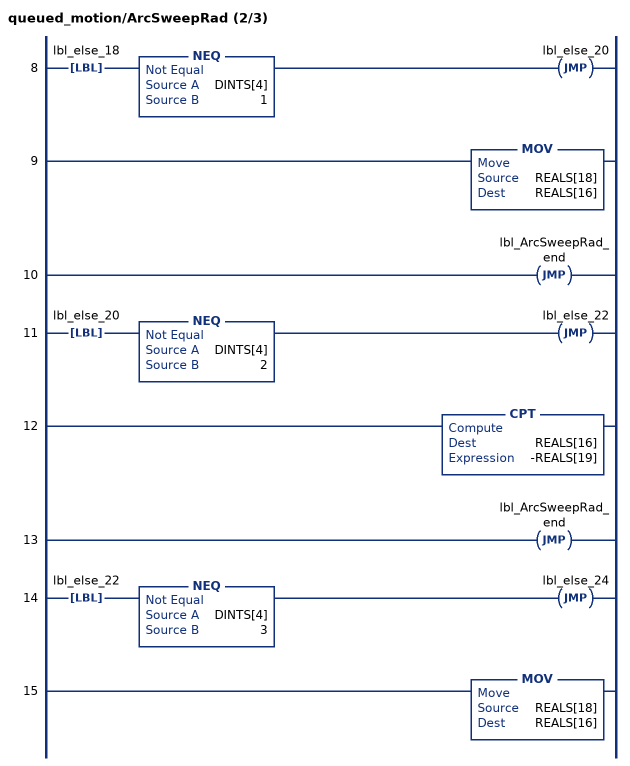
   8: LBL(lbl_else_18)NEQ(DINTS[4],1)JMP(lbl_else_20);
   9: MOV(REALS[18],REALS[16]);
   10: JMP(lbl_ArcSweepRad_end);
   11: LBL(lbl_else_20)NEQ(DINTS[4],2)JMP(lbl_else_22);
   12: CPT(REALS[16],-REALS[19]);
   13: JMP(lbl_ArcSweepRad_end);
   14: LBL(lbl_else_22)NEQ(DINTS[4],3)JMP(lbl_else_24);
   15: MOV(REALS[18],REALS[16]);
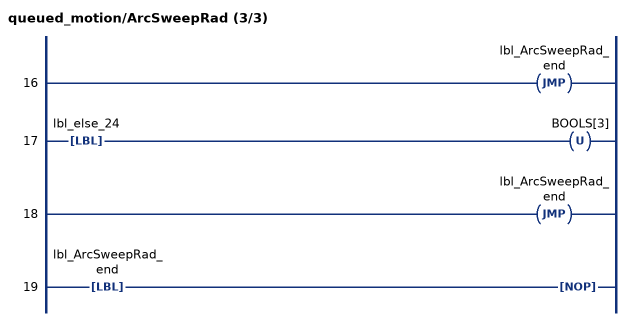
   16: JMP(lbl_ArcSweepRad_end);
   17: LBL(lbl_else_24)OTU(BOOLS[3]);
   18: JMP(lbl_ArcSweepRad_end);
   19: LBL(lbl_ArcSweepRad_end)NOP();
END_ROUTINE
